FUNCTION_BLOCK mySumFb
VAR_INPUT
	sum1,sum2:REAL;
END_VAR
VAR_OUTPUT
	result:real;
END_VAR
VAR
END_VAR

result := sum1+sum2;

END_FUNCTION_BLOCK

(* stored: Version 1.1.0.1, ProductVersion 3.1.4024.6
   POU mySumFb: Id {d6ea5f8e-d44f-4e52-a80f-9d3a013f6690}, SpecialFunc None *)
